(* IEC 61131-3 sources: com.logicals.lc3.webinar/usRTS_RPMControl_iSOC/src_FB_LIB_SAFE/Numeric/DINT, 8 files *)

(* ---- wADD_DINT_2.iecst ---- *)
NAMESPACE logicals.web.standard
NAMESPACE numeric

/*
 * Function block wrapper for IEC 61131-3 ADD<br>
 * IN1 =  1st value (DINT)<br>
 * IN2 =  2nd value (DINT)<br>
 * OUT = Sum of all input values (DINT)<br>
 */
FUNCTION_BLOCK wADD_DINT_2
	{ vNameAlignment:="center"; altName:="+"; bgColor:="LightPink"; width:=40; hideIONames; }
	VAR_INPUT
		IN1 : DINT;
		IN2 : DINT;
	END_VAR
	VAR_OUTPUT
		OUT : DINT;
	END_VAR

	OUT := ADD(IN1:=IN1, IN2:=IN2, ENO=>ENO);
END_FUNCTION_BLOCK

END_NAMESPACE
END_NAMESPACE

(* ---- wADD_DINT_3.iecst ---- *)
NAMESPACE logicals.web.standard
NAMESPACE numeric

/*
 * Function block wrapper for IEC 61131-3 ADD<br>
 * IN1 =  1st value (DINT)<br>
 * IN2 =  2nd value (DINT)<br>
 * IN3 =  3rd value (DINT)<br>
 * OUT = Sum of all input values (DINT)<br>
 */
FUNCTION_BLOCK wADD_DINT_3
	{ vNameAlignment:="center"; altName:="+"; bgColor:="LightPink"; width:=40; hideIONames; }
	VAR_INPUT
		IN1 : DINT;
		IN2 : DINT;
		IN3 : DINT;
	END_VAR
	VAR_OUTPUT
		OUT : DINT;
	END_VAR

	OUT := ADD(IN1:=IN1, IN2:=IN2, IN3:=IN3, ENO=>ENO);
END_FUNCTION_BLOCK

END_NAMESPACE
END_NAMESPACE

(* ---- wADD_DINT_4.iecst ---- *)
NAMESPACE logicals.web.standard
NAMESPACE numeric

/*
 * Function block wrapper for IEC 61131-3 ADD<br>
 * IN1 =  1st value (DINT)<br>
 * IN2 =  2nd value (DINT)<br>
 * IN3 =  3rd value (DINT)<br>
 * IN4 =  4th value (DINT)<br>
 * OUT = Sum of all input values (DINT)<br>
 */
FUNCTION_BLOCK wADD_DINT_4
	{ vNameAlignment:="center"; altName:="+"; bgColor:="LightPink"; width:=40; hideIONames; }
	VAR_INPUT
		IN1 : DINT;
		IN2 : DINT;
		IN3 : DINT;
		IN4 : DINT;
	END_VAR
	VAR_OUTPUT
		OUT : DINT;
	END_VAR

	OUT := ADD(IN1:=IN1, IN2:=IN2, IN3:=IN3, IN4:=IN4, ENO=>ENO);
END_FUNCTION_BLOCK

END_NAMESPACE
END_NAMESPACE

(* ---- wDIV_DINT.iecst ---- *)
NAMESPACE logicals.web.standard
NAMESPACE numeric

/*
 * Function block wrapper for IEC 61131-3 DIV<br>
 * IN1 =  1st value (DINT)<br>
 * IN2 =  2nd value (DINT)<br>
 * OUT = quotient of IN1 divided by IN2 (DINT)<br>
 */
FUNCTION_BLOCK wDIV_DINT
	{ vNameAlignment:="center"; altName:="/"; bgColor:="LightPink"; width:=40; hideIONames; }
	VAR_INPUT
		IN1 : DINT;
		IN2 : DINT;
	END_VAR
	VAR_OUTPUT
		OUT : DINT;
	END_VAR

	OUT := DIV(IN1:=IN1, IN2:=IN2, ENO=>ENO);
END_FUNCTION_BLOCK

END_NAMESPACE
END_NAMESPACE

(* ---- wMUL_DINT_2.iecst ---- *)
NAMESPACE logicals.web.standard
NAMESPACE numeric

/*
 * Function block wrapper for IEC 61131-3 MUL<br>
 * IN1 =  1st value (DINT)<br>
 * IN2 =  2nd value (DINT)<br>
 * OUT = Product of multiplication of all inputs (DINT)<br>
 */
FUNCTION_BLOCK wMUL_DINT_2
	{ vNameAlignment:="center"; altName:="*"; bgColor:="LightPink"; width:=40; hideIONames; }
	VAR_INPUT
		IN1 : DINT;
		IN2 : DINT;
	END_VAR
	VAR_OUTPUT
		OUT : DINT;
	END_VAR

	OUT := MUL(IN1:=IN1, IN2:=IN2, ENO=>ENO);
END_FUNCTION_BLOCK

END_NAMESPACE
END_NAMESPACE

(* ---- wMUL_DINT_3.iecst ---- *)
NAMESPACE logicals.web.standard
NAMESPACE numeric

/*
 * Function block wrapper for IEC 61131-3 MUL<br>
 * IN1 =  1st value (DINT)<br>
 * IN2 =  2nd value (DINT)<br>
 * IN3 =  3rd value (DINT)<br>
 * OUT = Product of multiplication of all inputs (DINT)<br>
 */
FUNCTION_BLOCK wMUL_DINT_3
	{ vNameAlignment:="center"; altName:="*"; bgColor:="LightPink"; width:=40; hideIONames; }
	VAR_INPUT
		IN1 : DINT;
		IN2 : DINT;
		IN3 : DINT;
	END_VAR
	VAR_OUTPUT
		OUT : DINT;
	END_VAR

	OUT := MUL(IN1:=IN1, IN2:=IN2, IN3:=IN3, ENO=>ENO);
END_FUNCTION_BLOCK

END_NAMESPACE
END_NAMESPACE

(* ---- wMUL_DINT_4.iecst ---- *)
NAMESPACE logicals.web.standard
NAMESPACE numeric

/*
 * Function block wrapper for IEC 61131-3 MUL<br>
 * IN1 =  1st value (DINT)<br>
 * IN2 =  2nd value (DINT)<br>
 * IN3 =  3rd value (DINT)<br>
 * IN4 =  4th value (DINT)<br>
 * OUT = Product of multiplication of all inputs (DINT)<br>
 */
FUNCTION_BLOCK wMUL_DINT_4
	{ vNameAlignment:="center"; altName:="*"; bgColor:="LightPink"; width:=40; hideIONames; }
	VAR_INPUT
		IN1 : DINT;
		IN2 : DINT;
		IN3 : DINT;
		IN4 : DINT;
	END_VAR
	VAR_OUTPUT
		OUT : DINT;
	END_VAR

	OUT := MUL(IN1:=IN1, IN2:=IN2, IN3:=IN3, IN4:=IN4, ENO=>ENO);
END_FUNCTION_BLOCK

END_NAMESPACE
END_NAMESPACE

(* ---- wSUB_DINT.iecst ---- *)
NAMESPACE logicals.web.standard
NAMESPACE numeric

/*
 * Function block wrapper for IEC 61131-3 SUB<br>
 * IN1 =  1st value (DINT)<br>
 * IN2 =  2nd value (DINT)<br>
 * OUT = IN1 minus IN2 (DINT)<br>
 */
FUNCTION_BLOCK wSUB_DINT
	{ vNameAlignment:="center"; altName:="-"; bgColor:="LightPink"; width:=40; hideIONames; }
	VAR_INPUT
		IN1 : DINT;
		IN2 : DINT;
	END_VAR
	VAR_OUTPUT
		OUT : DINT;
	END_VAR

	OUT := SUB(IN1:=IN1, IN2:=IN2, ENO=>ENO);
END_FUNCTION_BLOCK

END_NAMESPACE
END_NAMESPACE
